FUNCTION_BLOCK SimpleLogSource IMPLEMENTS I_SimpleLogSource
VAR
	{attribute 'hide'}
	_SourceName : T_MaxString;
	{attribute 'hide'}
	_TimeStamp : T_FILETIME64;
END_VAR

{attribute 'monitoring' := 'call'}
PROPERTY SourceName : T_MaxString
GET
SourceName := _SourceName;
END_GET
SET
_SourceName := SourceName;
END_SET
END_PROPERTY

{attribute 'monitoring' := 'call'}
PROPERTY TimeStamp : T_FILETIME64
GET
TimeStamp := _TimeStamp;
END_GET
SET
_TimeStamp := TimeStamp;
END_SET
END_PROPERTY

END_FUNCTION_BLOCK

(* stored: Version 1.1.0.1
   POU SimpleLogSource: Id {afe55241-3057-4122-abfb-57743fcfe2a9}, SpecialFunc None
   Property SourceName: Id {4a6a0d2d-b69f-47ba-824a-2c2cb7762739}
   Get Get: Id {7493dc3e-787e-4601-a8b3-94a3e75fae51}
   Set Set: Id {57a20b66-ae7a-4e9a-b3c7-c981f732ab73}
   Property TimeStamp: Id {0aa61d6c-284a-45c2-ad9c-1aa79e20be48}
   Get Get: Id {d8c5ad5e-95c2-4d7e-9edd-42f1f910325d}
   Set Set: Id {9959a51c-4a38-4905-830c-3ead4d403625} *)
